// TIA Portal V15.1 export
// export: Created 2024-05-17T05:38:59.0964494Z, ExportSetting WithDefaults, DisplayName Totally Integrated Automation Portal, DisplayVersion V15.1 Update 5, DisplayName TIA Portal Openness, DisplayVersion V15.1 Update 5, DisplayName SINAMICS Startdrive Advanced, DisplayVersion V15.1, DisplayName G130, G150, S120, S150, SINAMICS MV, S210, DisplayVersion V15.1, DisplayName G110M, G120, G120C, G120D, G120P, DisplayVersion V15.1, DisplayName STEP 7 Professional, DisplayVersion V15.1 Update 5, DisplayName STEP 7 Safety, DisplayVersion V15.1, DisplayName WinCC Professional, DisplayVersion V15.1 Update 5, DisplayName SIMATIC Visualization Architect, DisplayVersion V15.1
FUNCTION "209230ZM01Config" : Void   // FC402, FBD
TITLE = 209230ZM01 ModeZone Configuration
{ S7_Optimized_Access := 'FALSE' }
AUTHOR : VCC
VERSION : 0.1
// stored: AutoNumber false, IsIECCheckEnabled false, SetENOAutomatically False, UDAEnableTagReadback false
BEGIN

REGION Network 1: **** 4.2 - Machine Status - Parameters **** Andon
   // Andon Config VCG
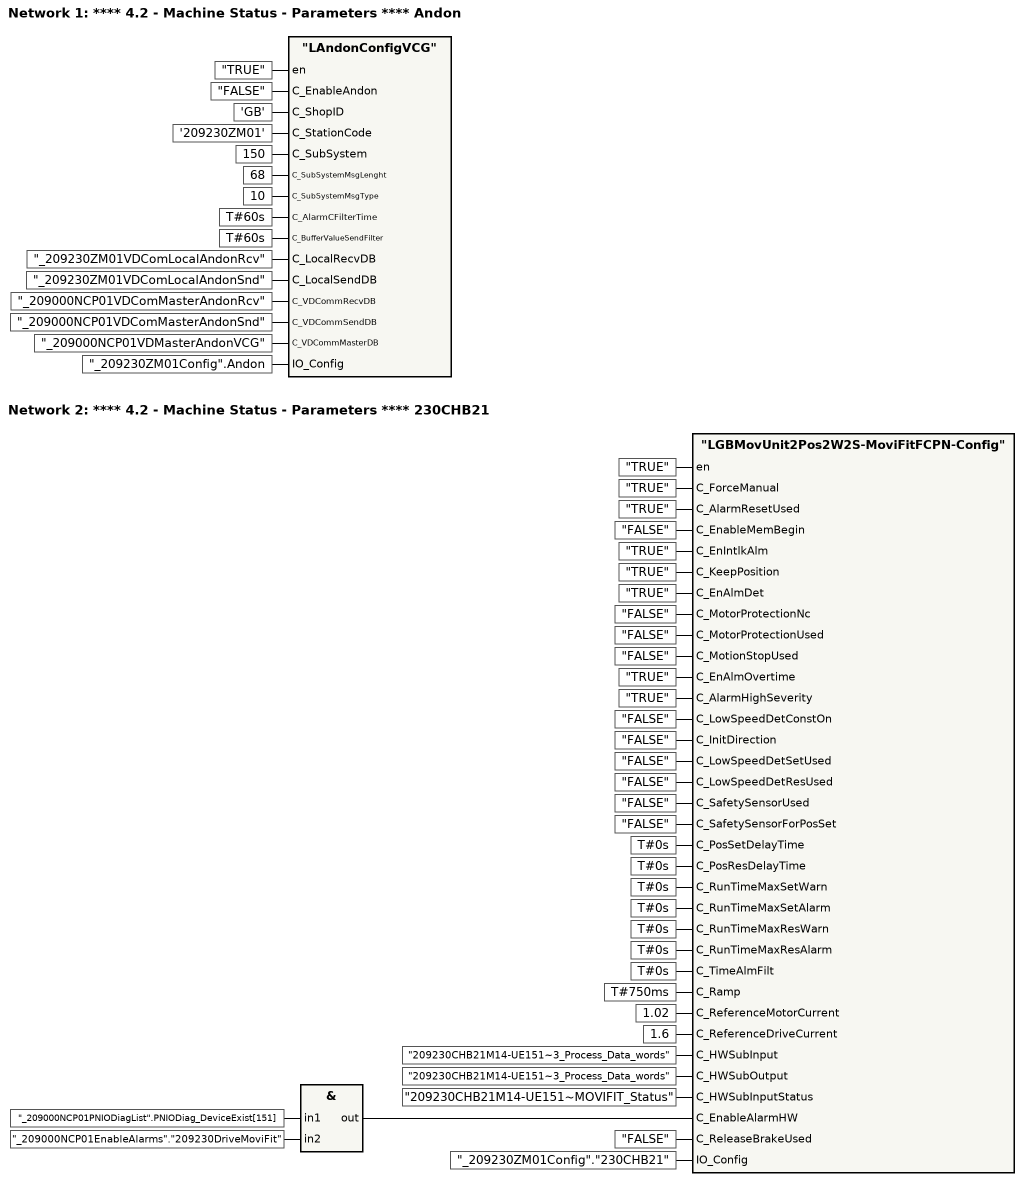
   IF "TRUE" THEN
       "LAndonConfigVCG"(C_EnableAndon := "FALSE",
                         C_ShopID := 'GB',
                         C_StationCode := '209230ZM01',
                         C_SubSystem := 150,
                         C_SubSystemMsgLenght := 68,
                         C_SubSystemMsgType := 10,
                         C_AlarmCFilterTime := T#60s,
                         C_BufferValueSendFilter := T#60s,
                         C_LocalRecvDB := "_209230ZM01VDComLocalAndonRcv",
                         C_LocalSendDB := "_209230ZM01VDComLocalAndonSnd",
                         C_VDCommRecvDB := "_209000NCP01VDComMasterAndonRcv",
                         C_VDCommSendDB := "_209000NCP01VDComMasterAndonSnd",
                         C_VDCommMasterDB := "_209000NCP01VDMasterAndonVCG",
                         IO_Config := "_209230ZM01Config".Andon);
   END_IF;
END_REGION

REGION Network 2: **** 4.2 - Machine Status - Parameters **** 230CHB21
   IF "TRUE" THEN
       "LGBMovUnit2Pos2W2S-MoviFitFCPN-Config"(C_ForceManual := "TRUE",
                               C_AlarmResetUsed := "TRUE",
                               C_EnableMemBegin := "FALSE",
                               C_EnIntlkAlm := "TRUE",
                               C_KeepPosition := "TRUE",
                               C_EnAlmDet := "TRUE",
                               C_MotorProtectionNc := "FALSE",
                               C_MotorProtectionUsed := "FALSE",
                               C_MotionStopUsed := "FALSE",
                               C_EnAlmOvertime := "TRUE",
                               C_AlarmHighSeverity := "TRUE",
                               C_LowSpeedDetConstOn := "FALSE",
                               C_InitDirection := "FALSE",
                               C_LowSpeedDetSetUsed := "FALSE",
                               C_LowSpeedDetResUsed := "FALSE",
                               C_SafetySensorUsed := "FALSE",
                               C_SafetySensorForPosSet := "FALSE",
                               C_PosSetDelayTime := T#0s,
                               C_PosResDelayTime := T#0s,
                               C_RunTimeMaxSetWarn := T#0s,
                               C_RunTimeMaxSetAlarm := T#0s,
                               C_RunTimeMaxResWarn := T#0s,
                               C_RunTimeMaxResAlarm := T#0s,
                               C_TimeAlmFilt := T#0s,
                               C_Ramp := T#750ms,
                               C_ReferenceMotorCurrent := 1.02,
                               C_ReferenceDriveCurrent := 1.6,
                               C_HWSubInput := "209230CHB21M14-UE151~3_Process_Data_words",
                               C_HWSubOutput := "209230CHB21M14-UE151~3_Process_Data_words",
                               C_HWSubInputStatus := "209230CHB21M14-UE151~MOVIFIT_Status",
                               C_EnableAlarmHW := "_209000NCP01PNIODiagList".PNIODiag_DeviceExist[151] AND "_209000NCP01EnableAlarms"."209230DriveMoviFit",
                               C_ReleaseBrakeUsed := "FALSE",
                               IO_Config := "_209230ZM01Config"."230CHB21");
   END_IF;
END_REGION

REGION Network 3: **** 4.2 - Machine Status - Parameters **** 230CHB22
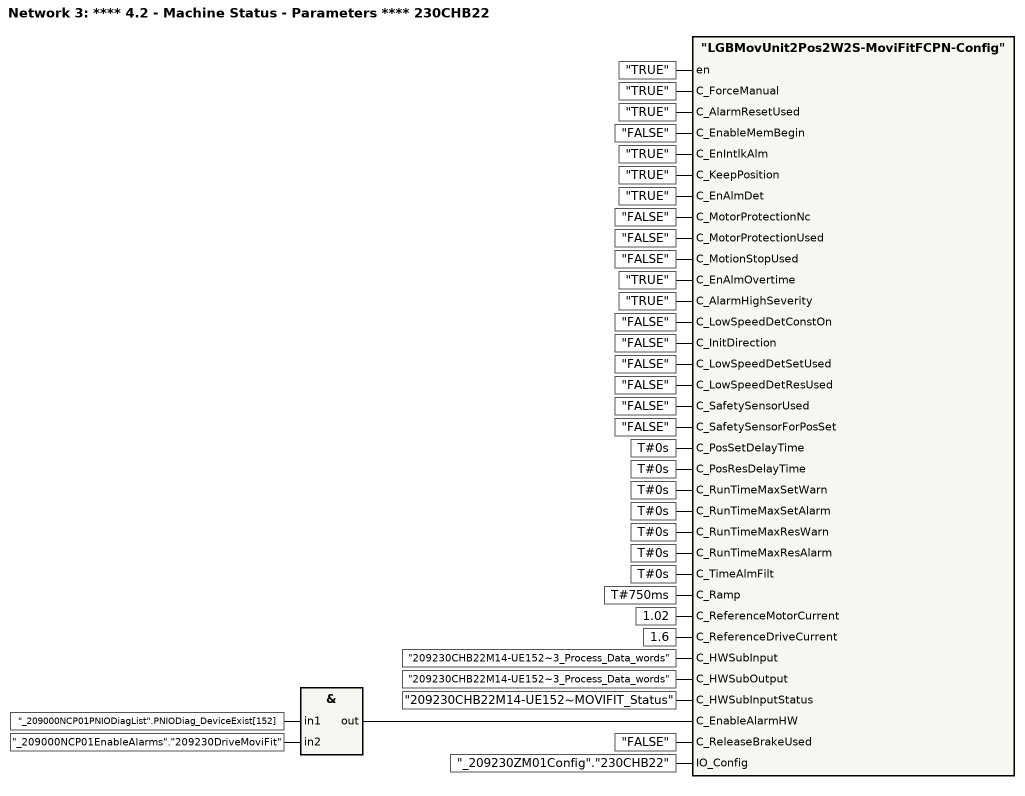
   IF "TRUE" THEN
       "LGBMovUnit2Pos2W2S-MoviFitFCPN-Config"(C_ForceManual := "TRUE",
                               C_AlarmResetUsed := "TRUE",
                               C_EnableMemBegin := "FALSE",
                               C_EnIntlkAlm := "TRUE",
                               C_KeepPosition := "TRUE",
                               C_EnAlmDet := "TRUE",
                               C_MotorProtectionNc := "FALSE",
                               C_MotorProtectionUsed := "FALSE",
                               C_MotionStopUsed := "FALSE",
                               C_EnAlmOvertime := "TRUE",
                               C_AlarmHighSeverity := "TRUE",
                               C_LowSpeedDetConstOn := "FALSE",
                               C_InitDirection := "FALSE",
                               C_LowSpeedDetSetUsed := "FALSE",
                               C_LowSpeedDetResUsed := "FALSE",
                               C_SafetySensorUsed := "FALSE",
                               C_SafetySensorForPosSet := "FALSE",
                               C_PosSetDelayTime := T#0s,
                               C_PosResDelayTime := T#0s,
                               C_RunTimeMaxSetWarn := T#0s,
                               C_RunTimeMaxSetAlarm := T#0s,
                               C_RunTimeMaxResWarn := T#0s,
                               C_RunTimeMaxResAlarm := T#0s,
                               C_TimeAlmFilt := T#0s,
                               C_Ramp := T#750ms,
                               C_ReferenceMotorCurrent := 1.02,
                               C_ReferenceDriveCurrent := 1.6,
                               C_HWSubInput := "209230CHB22M14-UE152~3_Process_Data_words",
                               C_HWSubOutput := "209230CHB22M14-UE152~3_Process_Data_words",
                               C_HWSubInputStatus := "209230CHB22M14-UE152~MOVIFIT_Status",
                               C_EnableAlarmHW := "_209000NCP01PNIODiagList".PNIODiag_DeviceExist[152] AND "_209000NCP01EnableAlarms"."209230DriveMoviFit",
                               C_ReleaseBrakeUsed := "FALSE",
                               IO_Config := "_209230ZM01Config"."230CHB22");
   END_IF;
END_REGION

REGION Network 4: **** 4.2 - Machine Status - Parameters **** 230CA21
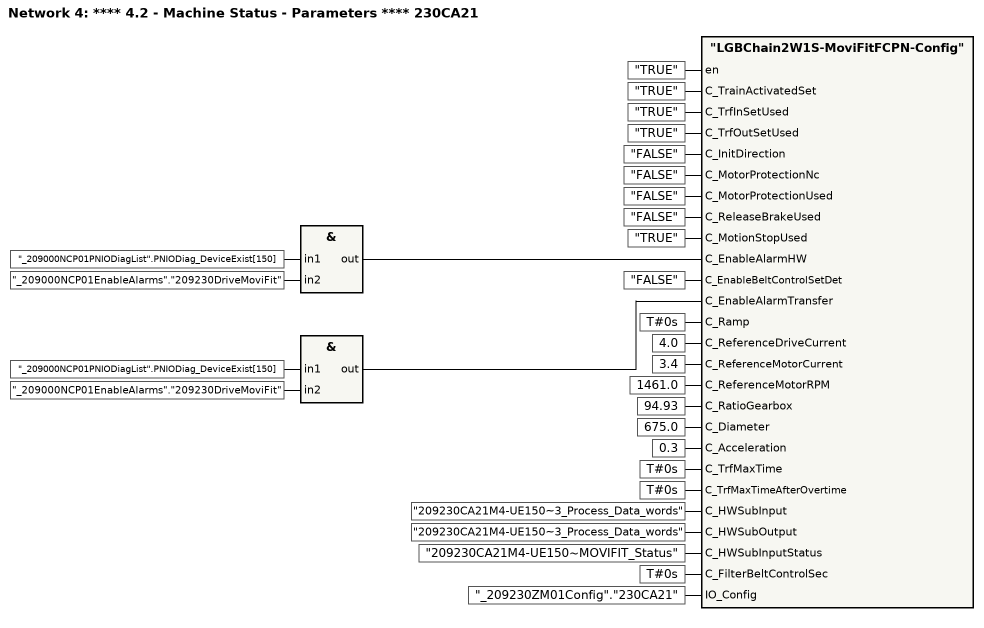
   IF "TRUE" THEN
       "LGBChain2W1S-MoviFitFCPN-Config"(C_TrainActivatedSet := "TRUE",
                               C_TrfInSetUsed := "TRUE",
                               C_TrfOutSetUsed := "TRUE",
                               C_InitDirection := "FALSE",
                               C_MotorProtectionNc := "FALSE",
                               C_MotorProtectionUsed := "FALSE",
                               C_ReleaseBrakeUsed := "FALSE",
                               C_MotionStopUsed := "TRUE",
                               C_EnableAlarmHW := "_209000NCP01PNIODiagList".PNIODiag_DeviceExist[150] AND "_209000NCP01EnableAlarms"."209230DriveMoviFit",
                               C_EnableBeltControlSetDet := "FALSE",
                               C_EnableAlarmTransfer := "_209000NCP01PNIODiagList".PNIODiag_DeviceExist[150] AND "_209000NCP01EnableAlarms"."209230DriveMoviFit",
                               C_Ramp := T#0s,
                               C_ReferenceDriveCurrent := 4.0,
                               C_ReferenceMotorCurrent := 3.4,
                               C_ReferenceMotorRPM := 1461.0,
                               C_RatioGearbox := 94.93,
                               C_Diameter := 675.0,
                               C_Acceleration := 0.3,
                               C_TrfMaxTime := T#0s,
                               C_TrfMaxTimeAfterOvertime := T#0s,
                               C_HWSubInput := "209230CA21M4-UE150~3_Process_Data_words",
                               C_HWSubOutput := "209230CA21M4-UE150~3_Process_Data_words",
                               C_HWSubInputStatus := "209230CA21M4-UE150~MOVIFIT_Status",
                               C_FilterBeltControlSec := T#0s,
                               IO_Config := "_209230ZM01Config"."230CA21");
   END_IF;
END_REGION

REGION Network 5: **** 4.2 - Machine Status - Parameters **** 230CR22
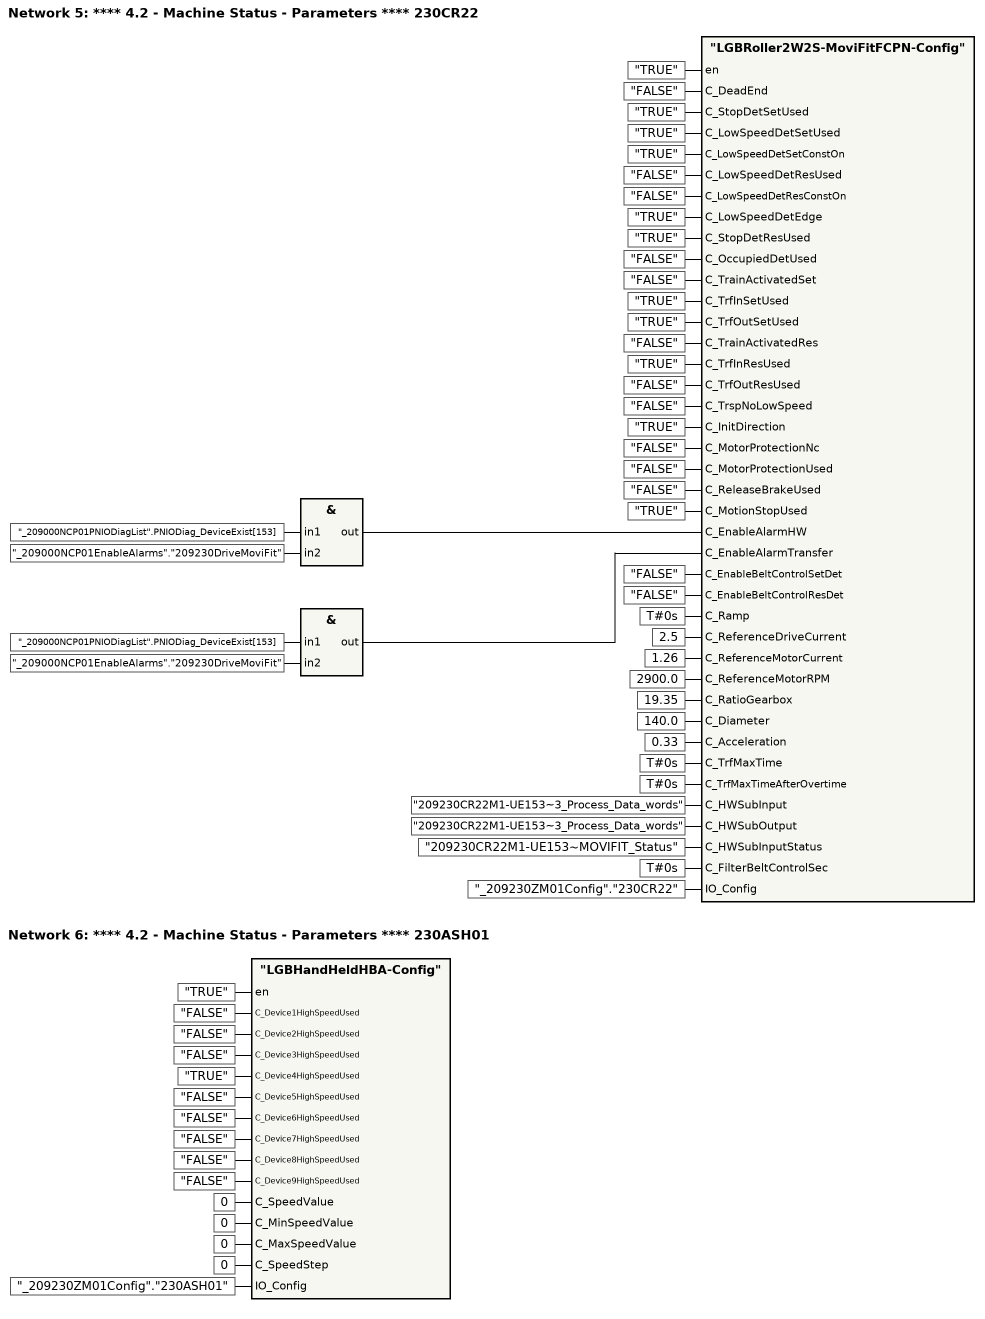
   IF "TRUE" THEN
       "LGBRoller2W2S-MoviFitFCPN-Config"(C_DeadEnd := "FALSE",
                               C_StopDetSetUsed := "TRUE",
                               C_LowSpeedDetSetUsed := "TRUE",
                               C_LowSpeedDetSetConstOn := "TRUE",
                               C_LowSpeedDetResUsed := "FALSE",
                               C_LowSpeedDetResConstOn := "FALSE",
                               C_LowSpeedDetEdge := "TRUE",
                               C_StopDetResUsed := "TRUE",
                               C_OccupiedDetUsed := "FALSE",
                               C_TrainActivatedSet := "FALSE",
                               C_TrfInSetUsed := "TRUE",
                               C_TrfOutSetUsed := "TRUE",
                               C_TrainActivatedRes := "FALSE",
                               C_TrfInResUsed := "TRUE",
                               C_TrfOutResUsed := "FALSE",
                               C_TrspNoLowSpeed := "FALSE",
                               C_InitDirection := "TRUE",
                               C_MotorProtectionNc := "FALSE",
                               C_MotorProtectionUsed := "FALSE",
                               C_ReleaseBrakeUsed := "FALSE",
                               C_MotionStopUsed := "TRUE",
                               C_EnableAlarmHW := "_209000NCP01PNIODiagList".PNIODiag_DeviceExist[153] AND "_209000NCP01EnableAlarms"."209230DriveMoviFit",
                               C_EnableAlarmTransfer := "_209000NCP01PNIODiagList".PNIODiag_DeviceExist[153] AND "_209000NCP01EnableAlarms"."209230DriveMoviFit",
                               C_EnableBeltControlSetDet := "FALSE",
                               C_EnableBeltControlResDet := "FALSE",
                               C_Ramp := T#0s,
                               C_ReferenceDriveCurrent := 2.5,
                               C_ReferenceMotorCurrent := 1.26,
                               C_ReferenceMotorRPM := 2900.0,
                               C_RatioGearbox := 19.35,
                               C_Diameter := 140.0,
                               C_Acceleration := 0.33,
                               C_TrfMaxTime := T#0s,
                               C_TrfMaxTimeAfterOvertime := T#0s,
                               C_HWSubInput := "209230CR22M1-UE153~3_Process_Data_words",
                               C_HWSubOutput := "209230CR22M1-UE153~3_Process_Data_words",
                               C_HWSubInputStatus := "209230CR22M1-UE153~MOVIFIT_Status",
                               C_FilterBeltControlSec := T#0s,
                               IO_Config := "_209230ZM01Config"."230CR22");
   END_IF;
END_REGION

REGION Network 6: **** 4.2 - Machine Status - Parameters **** 230ASH01
   IF "TRUE" THEN
       "LGBHandHeldHBA-Config"(C_Device1HighSpeedUsed := "FALSE",
                               C_Device2HighSpeedUsed := "FALSE",
                               C_Device3HighSpeedUsed := "FALSE",
                               C_Device4HighSpeedUsed := "TRUE",
                               C_Device5HighSpeedUsed := "FALSE",
                               C_Device6HighSpeedUsed := "FALSE",
                               C_Device7HighSpeedUsed := "FALSE",
                               C_Device8HighSpeedUsed := "FALSE",
                               C_Device9HighSpeedUsed := "FALSE",
                               C_SpeedValue := 0,
                               C_MinSpeedValue := 0,
                               C_MaxSpeedValue := 0,
                               C_SpeedStep := 0,
                               IO_Config := "_209230ZM01Config"."230ASH01");
   END_IF;
END_REGION
END_FUNCTION
